// Mitsubishi GX Works2 project: 9   PLC: FX2N/FX2NC

PROGRAM MAIN
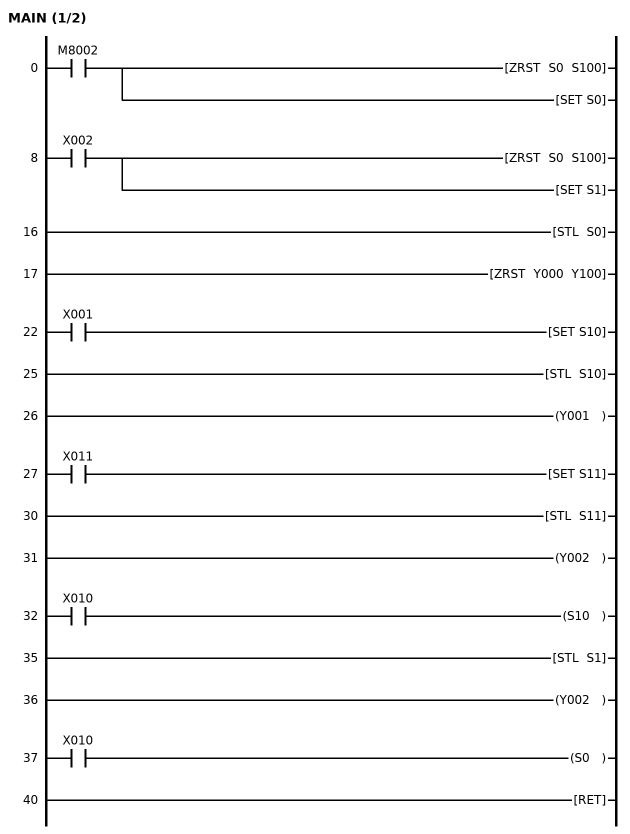
0     LD      M8002
      ZRST    S0 S100
      SET     S0
8     LD      X002
      ZRST    S0 S100
      SET     S1
16    STL     S0
17    ZRST    Y000 Y100
22    LD      X001
      SET     S10
25    STL     S10
26    OUT     Y001
27    LD      X011
      SET     S11
30    STL     S11
31    OUT     Y002
32    LD      X010
      OUT     S10
35    STL     S1
36    OUT     Y002
37    LD      X010
      OUT     S0
40    RET
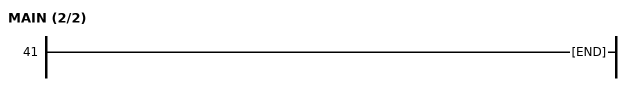
41    END
END_PROGRAM

// device comments not shown above
BL0  ; main
BL1  ; a
BL2  ; b
